FUNCTION_BLOCK EL5112
VAR
	_io : EL5112_Data;
	{attribute addProperty Name "WcState"}
	_wcState : WcStateInputToggle;
	{attribute addProperty Name "Info data"}
	_infoData : InfoDataAdsDC;
END_VAR

PROPERTY IO : REFERENCE TO EL5112_Data
GET
IO REF= _io;
END_GET
END_PROPERTY

PROPERTY WcState : REFERENCE TO WcStateInputToggle
GET
WcState REF= _wcState;
END_GET
END_PROPERTY

END_FUNCTION_BLOCK

(* stored: Version 1.1.0.1, ProductVersion 3.1.4024.9
   POU EL5112: Id {c253403c-6401-0413-2176-25df190be463}, SpecialFunc None
   Property IO: Id {424bbc33-3487-08ab-20bd-47b9cc895834}
   Get Get: Id {c94b07ee-a2d7-000c-02d6-dc4315436a57}
   Property WcState: Id {c247f607-1118-0b83-38ea-5f3735ea23e1}
   Get Get: Id {f004d7d0-03fa-0457-0b73-8a9df7734904} *)
